{attribute 'qualified_only'}
{attribute 'strict'}
{attribute 'to_string'}
TYPE EFoerderband :
(
	Off:=0,
	Init := 1,
	Ready := 2,
	Production := 3,
	Done := 4	
);
END_TYPE

(* stored: Version 1.1.0.1
   DUT EAnlageGes: Id {2a9a092b-f052-4d7d-93c4-4128ddd84c5c} *)
